FUNCTION DEG_TO_ARCSEC : LREAL
VAR_INPUT
    degrees : LREAL;
END_VAR
VAR
END_VAR

DEG_TO_ARCSEC := degrees * 3600.0;

END_FUNCTION

(* stored: Version 1.1.0.1, ProductVersion 3.1.4018.5
   POU DEG_TO_ARCSEC: Id {65fc53d6-3b68-4413-96b4-05b91c9bdb41}, SpecialFunc None *)
